{attribute 'linkalways'} 
{attribute 'no_explicit_call' := 'This FB is a CLASS and must be accessed using methods or properties'}
{attribute 'enable_dynamic_creation'}
FUNCTION_BLOCK FINAL ABS_UINT EXTENDS Node
VAR
	in : _UINT(0);
	out : _UINT(0);
END_VAR

METHOD PUBLIC Clone : I_Node
VAR
	pNode : POINTER TO ABS_UINT;
END_VAR
pNode := __NEW(ABS_UINT);
Clone := pNode^;
END_METHOD

METHOD FB_init : BOOL
VAR_INPUT
	bInitRetains : BOOL; // if TRUE, the retain variables are initialized (warm start / cold start)
	bInCopyCode : BOOL;  // if TRUE, the instance afterwards gets moved into the copy code (online change)
END_VAR
AddInput('in',THIS^.in);
AddOutput('out', THIS^.out);
END_METHOD

METHOD PROTECTED OnExecute
VAR
END_VAR
out.Value := ABS(in.Value);
END_METHOD

END_FUNCTION_BLOCK

(* stored: Version 1.1.0.1, ProductVersion 3.1.4024.15
   POU ABS_UINT: Id {5b34cea1-f30a-4b6f-b5f6-0141a1bd9a4b}, SpecialFunc None
   Folder Constructor: Id {3d31836b-b9fb-40fa-99b8-f8b39c2072a5}
   Method Clone: Id {86cfe524-7ca4-4302-966d-2cfb2029e29c}
   Method FB_init: Id {49ac6853-87b7-45d8-b65b-ff21499d82fb}
   Method OnExecute: Id {b0b1d28f-c0bf-437c-bc16-58b1ac623c2c} *)
